% RSLogix 500 project Project_4.RSS, saved by version 8.30.00.16 %
PROJECT "UNTITLED"    % processor: Bul.1763 MicroLogix 1100 Series B %

PROGRAM FILES
  LAD 2 "MAIN"  3 rungs
  LAD 3 "IO"  7 rungs
  LAD 4 "CONTROL"  11 rungs

DATA FILES
  O0 OUTPUT  5 elements
  I1 INPUT  7 elements
  S2 STATUS  66 elements
  B3 BINARY  2 elements
  T4 TIMER  3 elements
  C5 COUNTER  1 elements
  R6 CONTROL  1 elements
  N7 INTEGER  8 elements
  F8 FLOAT  1 elements
  N9 MOTOR  9 elements
  N10 CYCLE CONT  1 elements

LADDER 2 "MAIN"
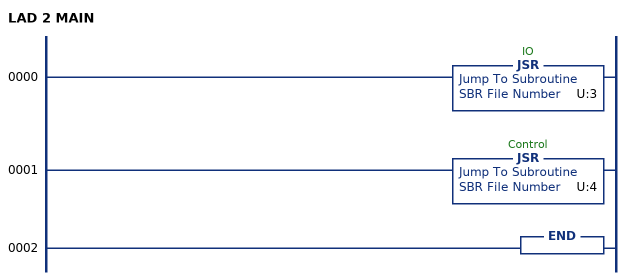
% Rung: 0 %
SOR JSR U:3 EOR
%   U:3  "IO" %
% Rung: 1 %
SOR JSR U:4 EOR
%   U:4  "Control" %
% Rung: 2 %
SOR END EOR

LADDER 3 "IO"
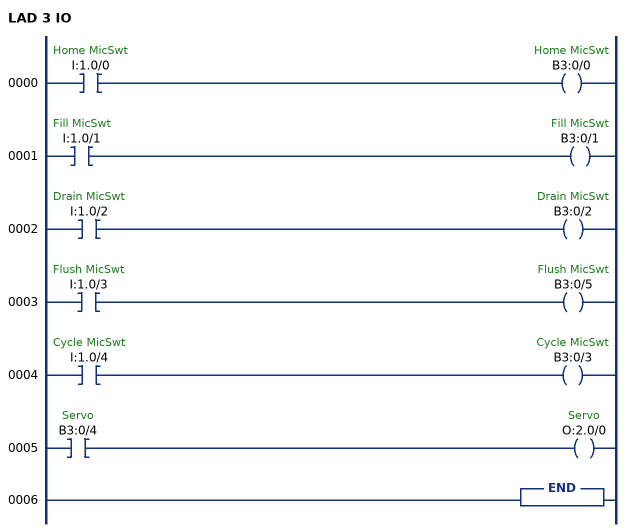
% Rung: 0 %
SOR XIC I:1.0/0 OTE B3:0/0 EOR
%   I:1.0/0  "Home MicSwt" %
%   B3:0/0  "Home MicSwt" %
% Rung: 1 %
SOR XIC I:1.0/1 OTE B3:0/1 EOR
%   I:1.0/1  "Fill MicSwt" %
%   B3:0/1  "Fill MicSwt" %
% Rung: 2 %
SOR XIC I:1.0/2 OTE B3:0/2 EOR
%   I:1.0/2  "Drain MicSwt" %
%   B3:0/2  "Drain MicSwt" %
% Rung: 3 %
SOR XIC I:1.0/3 OTE B3:0/5 EOR
%   I:1.0/3  "Flush MicSwt" %
%   B3:0/5  "Flush MicSwt" %
% Rung: 4 %
SOR XIC I:1.0/4 OTE B3:0/3 EOR
%   I:1.0/4  "Cycle MicSwt" %
%   B3:0/3  "Cycle MicSwt" %
% Rung: 5 %
SOR XIC B3:0/4 OTE O:2.0/0 EOR
%   B3:0/4  "Servo" %
%   O:2.0/0  "Servo" %
% Rung: 6 %
SOR END EOR

LADDER 4 "CONTROL"
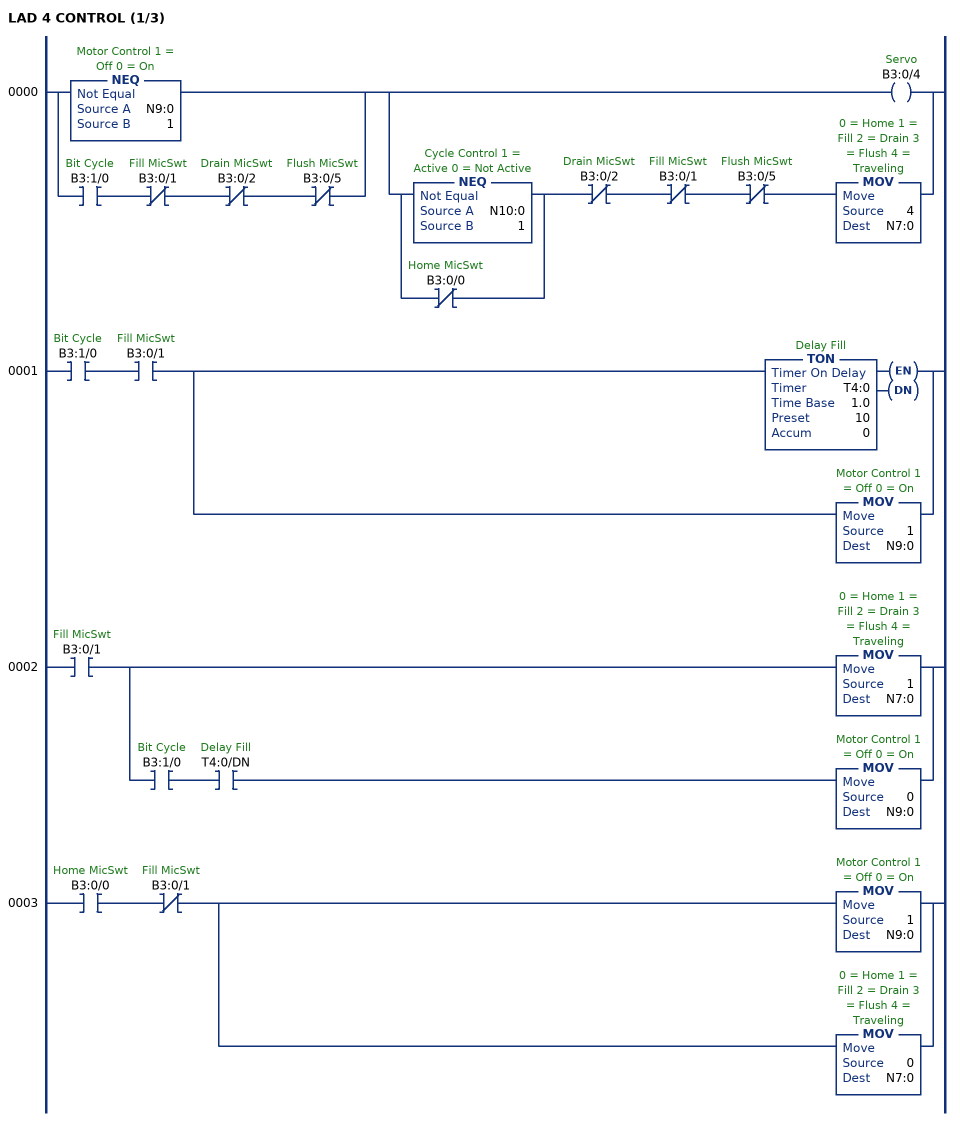
% Rung: 0 %
SOR BST NEQ N9:0 1 NXB XIC B3:1/0 XIO B3:0/1 XIO B3:0/2 XIO B3:0/5 BND BST OTE B3:0/4 NXB BST NEQ N10:0 1 NXB XIO B3:0/0 BND XIO B3:0/2 XIO B3:0/1 XIO B3:0/5 MOV 4 N7:0 BND EOR
%   N9:0  "Motor Control 1 = Off 0 = On" %
%   B3:1/0  "Bit Cycle" %
%   B3:0/1  "Fill MicSwt" %
%   B3:0/2  "Drain MicSwt" %
%   B3:0/5  "Flush MicSwt" %
%   B3:0/4  "Servo" %
%   N10:0  "Cycle Control 1 = Active 0 = Not Active" %
%   B3:0/0  "Home MicSwt" %
%   N7:0  "0 = Home 1 = Fill 2 = Drain 3 = Flush 4 = Traveling" %
% Rung: 1 %
SOR XIC B3:1/0 XIC B3:0/1 BST TON T4:0 1.0 10 0 NXB MOV 1 N9:0 BND EOR
%   B3:1/0  "Bit Cycle" %
%   B3:0/1  "Fill MicSwt" %
%   T4:0  "Delay Fill" %
%   N9:0  "Motor Control 1 = Off 0 = On" %
% Rung: 2 %
SOR XIC B3:0/1 BST MOV 1 N7:0 NXB XIC B3:1/0 XIC T4:0/DN MOV 0 N9:0 BND EOR
%   B3:0/1  "Fill MicSwt" %
%   N7:0  "0 = Home 1 = Fill 2 = Drain 3 = Flush 4 = Traveling" %
%   B3:1/0  "Bit Cycle" %
%   T4:0/DN  "Delay Fill" %
%   N9:0  "Motor Control 1 = Off 0 = On" %
% Rung: 3 %
SOR XIC B3:0/0 XIO B3:0/1 BST MOV 1 N9:0 NXB MOV 0 N7:0 BND EOR
%   B3:0/0  "Home MicSwt" %
%   B3:0/1  "Fill MicSwt" %
%   N9:0  "Motor Control 1 = Off 0 = On" %
%   N7:0  "0 = Home 1 = Fill 2 = Drain 3 = Flush 4 = Traveling" %

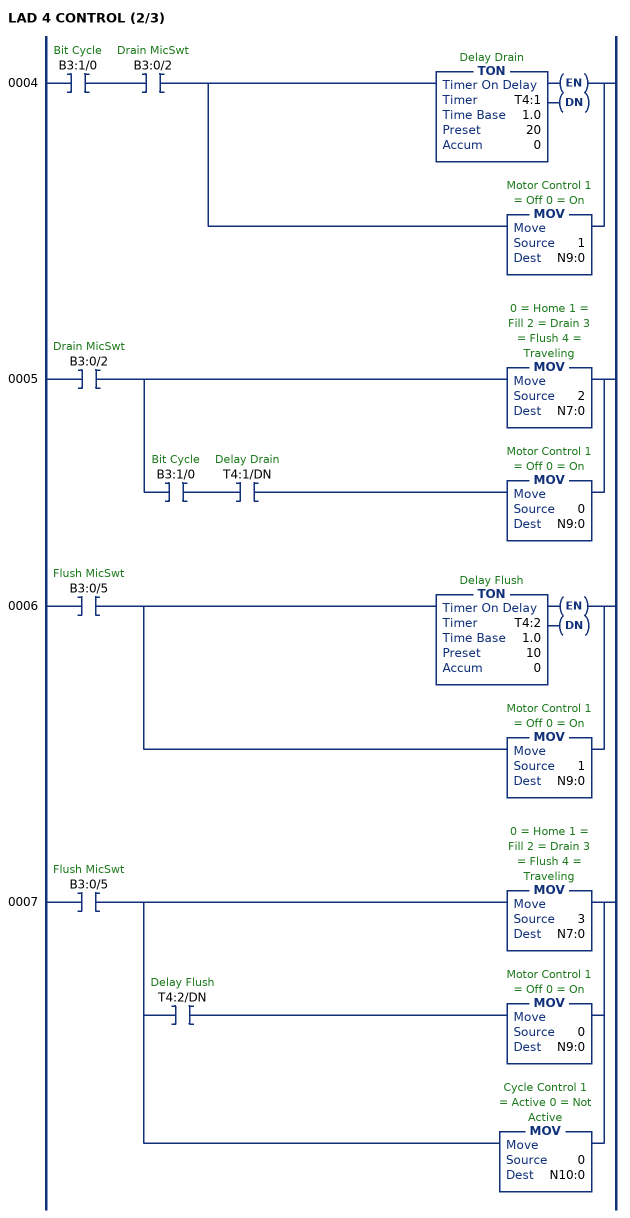
% Rung: 4 %
SOR XIC B3:1/0 XIC B3:0/2 BST TON T4:1 1.0 20 0 NXB MOV 1 N9:0 BND EOR
%   B3:1/0  "Bit Cycle" %
%   B3:0/2  "Drain MicSwt" %
%   T4:1  "Delay Drain" %
%   N9:0  "Motor Control 1 = Off 0 = On" %
% Rung: 5 %
SOR XIC B3:0/2 BST MOV 2 N7:0 NXB XIC B3:1/0 XIC T4:1/DN MOV 0 N9:0 BND EOR
%   B3:0/2  "Drain MicSwt" %
%   N7:0  "0 = Home 1 = Fill 2 = Drain 3 = Flush 4 = Traveling" %
%   B3:1/0  "Bit Cycle" %
%   T4:1/DN  "Delay Drain" %
%   N9:0  "Motor Control 1 = Off 0 = On" %
% Rung: 6 %
SOR XIC B3:0/5 BST TON T4:2 1.0 10 0 NXB MOV 1 N9:0 BND EOR
%   B3:0/5  "Flush MicSwt" %
%   T4:2  "Delay Flush" %
%   N9:0  "Motor Control 1 = Off 0 = On" %
% Rung: 7 %
SOR XIC B3:0/5 BST MOV 3 N7:0 NXB XIC T4:2/DN MOV 0 N9:0 NXB MOV 0 N10:0 BND EOR
%   B3:0/5  "Flush MicSwt" %
%   N7:0  "0 = Home 1 = Fill 2 = Drain 3 = Flush 4 = Traveling" %
%   T4:2/DN  "Delay Flush" %
%   N9:0  "Motor Control 1 = Off 0 = On" %
%   N10:0  "Cycle Control 1 = Active 0 = Not Active" %

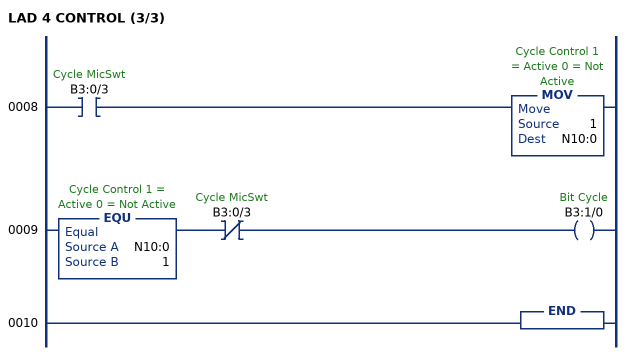
% Rung: 8 %
SOR XIC B3:0/3 MOV 1 N10:0 EOR
%   B3:0/3  "Cycle MicSwt" %
%   N10:0  "Cycle Control 1 = Active 0 = Not Active" %
% Rung: 9 %
SOR EQU N10:0 1 XIO B3:0/3 OTE B3:1/0 EOR
%   N10:0  "Cycle Control 1 = Active 0 = Not Active" %
%   B3:0/3  "Cycle MicSwt" %
%   B3:1/0  "Bit Cycle" %
% Rung: 10 %
SOR END EOR

OTHER DOCUMENTED ADDRESSES
  B3:1/1  "Bit Fill Servo"
  B3:1/2  "Bit Drain Servo"
  B3:1/3  "Bit Cycle Servo"
  B3:1/4  "Bit Flush Servo"
  B3:1/5  "Initiate"
  N7:1  "Servo Position"
  N7:7  "Initiate"
  N7:10  "Cycle Control 1 = Active 0 = Not Active"

DATA TABLE (non-zero values as saved)
DATA T4
% .PRE .ACC %
% T4:0 % 10 0
% T4:1 % 20 0
% T4:2 % 10 0
